KUKA KRL program: panpick_dry.src, panpick_dry.dat

--- panpick_dry.src ---
&ACCESS RVO1
&REL 107
&PARAM EDITMASK = *
&PARAM TEMPLATE = C:\KRC\Roboter\Template\vorgabe
&PARAM DISKPATH = KRC:\R1\Program\Sub Programs
DEF panpick_dry( )
;FOLD INI;%{PE}
  ;FOLD BASISTECH INI
    GLOBAL INTERRUPT DECL 3 WHEN $STOPMESS==TRUE DO IR_STOPM ( )
    INTERRUPT ON 3
    BAS (#INITMOV,0 )
  ;ENDFOLD (BASISTECH INI)
  ;FOLD USER INI
    ;Make your modifications here
INPICKER_Handler.DataToSend.command=0
 wait for (INPICKER_Handler.DataReceived.state==0)
REINTENTO=FALSE
;CILS_INIT()
  ;ENDFOLD (USER INI)
;ENDFOLD (INI)

if false then
;POS FOTO 1
;FOLD PTP P03 Vel=100 % PDAT1 Tool[0] Base[0];%{PE}%R 8.3.48,%MKUKATPBASIS,%CMOVE,%VPTP,%P 1:PTP, 2:P03, 3:, 5:100, 7:PDAT1
$BWDSTART=FALSE
PDAT_ACT=PPDAT1
FDAT_ACT=FP03
BAS(#PTP_PARAMS,100)
PTP XP03
;ENDFOLD
endif
INICIOFOTO:

;fold espera foto

IF ((POSBAT>0) AND (POSBAT<5)) THEN
 INPICKER_Handler.DataToSend.partid=3
ELSE
 INPICKER_Handler.DataToSend.partid=2
ENDIF
 INPICKER_Handler.DataToSend.command=1
 wait for (INPICKER_Handler.DataReceived.state==30)
 wait sec 0.5

;ENDFOLD

;EVALUA foto

IF (INPICKER_Handler.DataReceived.ObjectsGraspable>0)THEN



;FOLD CARGA FRAMEXP01
;FOTO OK
FRAMEAUX={X 0,Y 0,Z 0,A 0,B 0,C 0}
FRAMEAUX=INPICKER_Handler.DataReceived.PartsToGrasp0.Position
XP01.x=(FRAMEAUX.x/10)-2
XP01.y=(FRAMEAUX.y/10)
XP01.z=(FRAMEAUX.z/10)
XP01.a=(FRAMEAUX.a/10)
XP01.b=FRAMEAUX.b/10
XP01.c=FRAMEAUX.c/10
;ENDFOLD

;FOLD CARGA FRAME XP02
FRAMEAUX={X 0,Y 0,Z 0,A 0,B 0,C 0}
FRAMEAUX=INPICKER_Handler.DataReceived.PartsToGrasp0.PreGrasp0
XP02.x=(FRAMEAUX.x/10)-2
XP02.y=(FRAMEAUX.y/10)
XP02.z=(FRAMEAUX.z/10)
XP02.a=(FRAMEAUX.a/10)
XP02.b=FRAMEAUX.b/10
XP02.c=FRAMEAUX.c/10
;ENDFOLD


ELSE

IF (REINTENTO==FALSE) THEN
REINTENTO=TRUE
INPICKER_Handler.DataToSend.command=0
wait for (INPICKER_Handler.DataReceived.state==0)
GOTO INICIOFOTO
ENDIF

;FOTO NOK
if false then
;FOLD Fordtech.Tool_Req Tool Request: 1 ;%{PE}%MKUKATPUSER

Tool_Req (1)

;ENDFOLD
;FOLD Fordtech.Wait_Tool_Ready Wait Tool Ready: 1 ;%{PE}%MKUKATPUSER

Wait_Tool_Ready (1)

;ENDFOLD
endif
BACKJUMP=TRUE
GOTO PEXIT
ENDIF





;FOLD PTP P02 CONT Vel=100 % PDAT2 Tool[5] Base[0];%{PE}%R 8.3.48,%MKUKATPBASIS,%CMOVE,%VPTP,%P 1:PTP, 2:P02, 3:C_DIS, 5:100, 7:PDAT2
$BWDSTART=FALSE
PDAT_ACT=PPDAT2
FDAT_ACT=FP02
BAS(#PTP_PARAMS,100)
PTP XP02 C_DIS
;ENDFOLD



;FOLD LIN P01 Vel=2 m/s CPDAT3 Tool[5] Base[0];%{PE}%R 8.3.48,%MKUKATPBASIS,%CMOVE,%VLIN,%P 1:LIN, 2:P01, 3:, 5:2, 7:CPDAT3
$BWDSTART=FALSE
LDAT_ACT=LCPDAT3
FDAT_ACT=FP01
BAS(#CP_PARAMS,2)
LIN XP01
;ENDFOLD
;halt
CIL_BAT_ACTIVO()

;FOLD WAIT Time=2 sec;%{PE}%R 8.3.48,%MKUKATPBASIS,%CWAIT,%VWAIT,%P 3:2
WAIT SEC 2
;ENDFOLD
lin_rel {z 20}
PART_CHECK()
lin_rel {z -20}
CIL_BAT_REPOSO()
PART_CHECK_OFF()
INPICKER_Handler.DataToSend.command=0

lin_rel {z 20}

;fold P04

FRAMEAUX={X 0,Y 0,Z 0,A 0,B 0,C 0}
XP04=FRAMEAUX
XP04.x=XP02.x
XP04.y=XP02.y
XP04.z=(XP02.z)+110
XP04.a=XP02.a
XP04.b=XP02.b
XP04.c=XP02.c

;ENDFOLD

;FOLD PTP p04 CONT Vel=100 % PDAT4 Tool[5] Base[0];%{PE}%R 8.3.48,%MKUKATPBASIS,%CMOVE,%VPTP,%P 1:PTP, 2:p04, 3:C_DIS, 5:100, 7:PDAT4
$BWDSTART=FALSE
PDAT_ACT=PPDAT4
FDAT_ACT=Fp04
BAS(#PTP_PARAMS,100)
PTP Xp04 C_DIS
;ENDFOLD


;FOLD SYN OUT 41 'Job Ready 1' State=TRUE at START Delay=0 ms;%{PE}%R 8.3.48,%MKUKATPBASIS,%COUT,%VSYNOUT,%P 2:41, 3:Job Ready 1, 5:TRUE, 7:0, 9:0, 12:0
TRIGGER WHEN DISTANCE=0 DELAY=0 DO $OUT[41]=TRUE
;ENDFOLD



PEXIT:
END

--- panpick_dry.dat ---
&ACCESS RVO1
&REL 107
&PARAM EDITMASK = *
&PARAM TEMPLATE = C:\KRC\Roboter\Template\vorgabe
&PARAM DISKPATH = KRC:\R1\Program\Sub Programs
DEFDAT  panpick_dry
;FOLD EXTERNAL DECLARATIONS;%{PE}%MKUKATPBASIS,%CEXT,%VCOMMON,%P
;FOLD BASISTECH EXT;%{PE}%MKUKATPBASIS,%CEXT,%VEXT,%P
EXT  BAS (BAS_COMMAND  :IN,REAL  :IN )
DECL INT SUCCESS
;ENDFOLD (BASISTECH EXT)
;FOLD USER EXT;%{E}%MKUKATPUSER,%CEXT,%VEXT,%P
;Make your modifications here

;ENDFOLD (USER EXT)
;ENDFOLD (EXTERNAL DECLARATIONS)
DECL E6POS XP01={X 459.400,Y 1980.30,Z 705.200,A 270.200,B 0.700000,C 180.000}
DECL FDAT FP01={TOOL_NO 5,BASE_NO 0,IPO_FRAME #BASE,POINT2[] " "}
DECL PDAT PPDAT01={VEL 100.000,ACC 100.000,APO_DIST 500.000,APO_MODE #CDIS,GEAR_JERK 100.000,EXAX_IGN 0}
DECL MODULEPARAM_T LAST_TP_PARAMS={PARAMS[] "Kuka.VelocityFieldEnabled=True; Kuka.ColDetectFieldEnabled=True; Kuka.MovementParameterFieldEnabled=True; Kuka.IsAngleEnabled=False; Kuka.PointName=P02; Kuka.FrameData.base_no=0; Kuka.FrameData.tool_no=5; Kuka.FrameData.ipo_frame=#BASE; Kuka.isglobalpoint=False; Kuka.MoveDataPtpName=PDAT02; Kuka.MovementDataPdat.apo_mode=#CDIS; Kuka.MovementDataPdat.apo_dist=500; Kuka.MovementData.vel=2; Kuka.MovementData.acc=100; Kuka.MovementData.exax_ign=0; Kuka.VelocityPtp=100; Kuka.BlendingEnabled=False; Kuka.APXEnabled=False; Kuka.CurrentCDSetIndex=0; Kuka.FrameData.point2=; Kuka.MoveDataName=CPDAT2; Kuka.MovementData.cb={AUX_PT {ORI #CONSIDER,E1 #CONSIDER,E2 #CONSIDER,E3 #CONSIDER,E4 #CONSIDER,E5 #CONSIDER,E6 #CONSIDER},TARGET_PT {ORI #INTERPOLATE,E1 #INTERPOLATE,E2 #INTERPOLATE,E3 #INTERPOLATE,E4 #INTERPOLATE,E5 #INTERPOLATE,E6 #INTERPOLATE}}; Kuka.MovementData.apo_fac=50; Kuka.MovementData.apo_dist=500; Kuka.MovementData.axis_acc=100; Kuka.MovementData.axis_vel=100; Kuka.MovementData.circ_typ=#BASE; Kuka.MovementData.jerk_fac=50; Kuka.MovementData.ori_typ=#VAR; Kuka.VelocityPath=2                          "}
DECL E6POS XP02={X 459.300,Y 1979.70,Z 755.200,A 270.200,B 0.700000,C 180.000}
DECL FDAT FP02={TOOL_NO 5,BASE_NO 0,IPO_FRAME #BASE,POINT2[] " "}
DECL PDAT PPDAT02={VEL 100.000,ACC 100.000,APO_DIST 500.000,APO_MODE #CDIS,GEAR_JERK 100.000,EXAX_IGN 0}
DECL LDAT LCPDAT1={VEL 2.00000,ACC 100.000,APO_DIST 500.000,APO_FAC 50.0000,AXIS_VEL 100.000,AXIS_ACC 100.000,ORI_TYP #VAR,CIRC_TYP #BASE,JERK_FAC 50.0000,GEAR_JERK 100.000,EXAX_IGN 0,CB {AUX_PT {ORI #CONSIDER,E1 #CONSIDER,E2 #CONSIDER,E3 #CONSIDER,E4 #CONSIDER,E5 #CONSIDER,E6 #CONSIDER},TARGET_PT {ORI #INTERPOLATE,E1 #INTERPOLATE,E2 #INTERPOLATE,E3 #INTERPOLATE,E4 #INTERPOLATE,E5 #INTERPOLATE,E6 #INTERPOLATE}}}
DECL E6POS XP03={X 469.006378,Y 724.797424,Z 1470.31934,A -86.9976196,B 22.0779018,C -179.006119,S 6,T 27,E1 0.0,E2 0.0,E3 0.0,E4 0.0,E5 0.0,E6 0.0}
DECL FDAT FP03={TOOL_NO 0,BASE_NO 0,IPO_FRAME #BASE,POINT2[] " "}
DECL PDAT PPDAT03={VEL 100.000,ACC 100.000,APO_DIST 500.000,APO_MODE #CDIS,GEAR_JERK 100.000,EXAX_IGN 0}
DECL E6POS XP04={X 444.700,Y 1789.20,Z 972.100,A 267.700,B 0.100000,C 180.300}
DECL FDAT FP04={TOOL_NO 5,BASE_NO 0,IPO_FRAME #BASE,POINT2[] " ",TQ_STATE FALSE}
DECL PDAT PPDAT04={VEL 100.000,ACC 100.000,APO_DIST 500.000,APO_MODE #CDIS,GEAR_JERK 100.000,EXAX_IGN 0}
DECL E6POS XP1={X 2856.00,Y 12860.0,Z 6727.00,A 2708.00,B 8.00000,C 1797.00}
DECL E6POS XP2={X 2856.00,Y 12860.0,Z 6727.00,A 2708.00,B 8.00000,C 1797.00}
DECL E6POS XP3={X 2856.00,Y 12860.0,Z 6727.00,A 2708.00,B 8.00000,C 1797.00}
DECL E6POS XP05={X 284.000,Y 1258.50,Z 983.400,A 271.300,B 0.800000,C 179.700,S 0,T 0,E1 0.0,E2 0.0,E3 0.0,E4 0.0,E5 0.0,E6 0.0}
DECL FDAT FP05={TOOL_NO 5,BASE_NO 0,IPO_FRAME #BASE,POINT2[] " "}
DECL PDAT PPDAT05={VEL 100.000,ACC 100.000,APO_DIST 500.000,APO_MODE #CDIS,GEAR_JERK 100.000,EXAX_IGN 0}
DECL LDAT LCPDAT2={VEL 2.00000,ACC 100.000,APO_DIST 500.000,APO_FAC 50.0000,AXIS_VEL 100.000,AXIS_ACC 100.000,ORI_TYP #VAR,CIRC_TYP #BASE,JERK_FAC 50.0000,GEAR_JERK 100.000,EXAX_IGN 0,CB {AUX_PT {ORI #CONSIDER,E1 #CONSIDER,E2 #CONSIDER,E3 #CONSIDER,E4 #CONSIDER,E5 #CONSIDER,E6 #CONSIDER},TARGET_PT {ORI #INTERPOLATE,E1 #INTERPOLATE,E2 #INTERPOLATE,E3 #INTERPOLATE,E4 #INTERPOLATE,E5 #INTERPOLATE,E6 #INTERPOLATE}}}
DECL BASIS_SUGG_T LAST_BASIS={POINT1[] "P0                      ",POINT2[] "P0                      ",CP_PARAMS[] "CPDAT0                  ",PTP_PARAMS[] "PDAT0                   ",CONT[] "                        ",CP_VEL[] "2                       ",PTP_VEL[] " 100                    ",SYNC_PARAMS[] "SYNCDAT                 ",SPL_NAME[] "S0                      ",A_PARAMS[] "ADAT0                   "}
DECL PDAT PPDAT1={VEL 100.000,ACC 100.000,APO_DIST 100.000,GEAR_JERK 50.0000,EXAX_IGN 0}
DECL PDAT PPDAT2={VEL 100.000,ACC 100.000,APO_DIST 100.000,APO_MODE #CDIS,GEAR_JERK 50.0000,EXAX_IGN 0}
DECL LDAT LCPDAT3={VEL 2.00000,ACC 100.000,APO_DIST 100.000,APO_FAC 50.0000,AXIS_VEL 100.000,AXIS_ACC 100.000,ORI_TYP #VAR,CIRC_TYP #BASE,JERK_FAC 50.0000,GEAR_JERK 50.0000,EXAX_IGN 0}
DECL LDAT LCPDAT4={VEL 2.00000,ACC 100.000,APO_DIST 100.000,APO_FAC 50.0000,AXIS_VEL 100.000,AXIS_ACC 100.000,ORI_TYP #VAR,CIRC_TYP #BASE,JERK_FAC 50.0000,GEAR_JERK 50.0000,EXAX_IGN 0}
DECL E6POS XP4={X 290.951233,Y 816.177124,Z 1275.55042,A -86.9976196,B 22.0779018,C -179.006119,S 6,T 27,E1 0.0,E2 0.0,E3 0.0,E4 0.0,E5 0.0,E6 0.0}
DECL FDAT FP4={TOOL_NO 5,BASE_NO 0,IPO_FRAME #BASE,POINT2[] " ",TQ_STATE FALSE}
DECL PDAT PPDAT3={VEL 100.000,ACC 100.000,APO_DIST 100.000,APO_MODE #CDIS,GEAR_JERK 50.0000,EXAX_IGN 0}
DECL PDAT PPDAT4={VEL 100.000,ACC 100.000,APO_DIST 100.000,APO_MODE #CDIS,GEAR_JERK 50.0000,EXAX_IGN 0}
DECL E6POS XP5={X 442.124359,Y -682.465210,Z 1416.05603,A -171.206314,B 14.8656197,C -154.747955,S 6,T 26,E1 0.0,E2 0.0,E3 0.0,E4 0.0,E5 0.0,E6 0.0}
DECL FDAT FP5={TOOL_NO 5,BASE_NO 0,IPO_FRAME #BASE,POINT2[] " ",TQ_STATE FALSE}
DECL PDAT PPDAT5={VEL 100.000,ACC 100.000,APO_DIST 100.000,APO_MODE #CDIS,GEAR_JERK 50.0000,EXAX_IGN 0}
ENDDAT
